// TIA Portal V18 export
// export: Created 2026-01-09T11:31:59.9051336Z, ExportSetting WithDefaults, DisplayName Totally Integrated Automation Portal, DisplayVersion V18 Update 5, DisplayName TIA Portal Openness, DisplayVersion V18 Update 5, DisplayName TIA Portal Teamcenter Gateway, DisplayVersion V18, DisplayName TIA Portal Version Control Interface, DisplayVersion V18, DisplayName SINAMICS Startdrive Advanced, DisplayVersion V18 SP2 Update 1, DisplayName SINAMICS Startdrive G110M, G120, G120C, G120D, G120P, G115D, DisplayVersion V18 SP2 Update 1, DisplayName SINAMICS Startdrive G130, G150, S120, S150, SINAMICS MV, S210, G220, S200, DisplayVersion V18 SP2 Update 1, DisplayName STEP 7 Professional, DisplayVersion V18 Update 5, DisplayName STEP 7 Safety, DisplayVersion V18, DisplayName WinCC Professional, DisplayVersion V18 Update 5
TagTable "1Command PLC To Mes_DB500"
  PLCtoMES_Load_Station1ChickInReq : Bool  (PLC tag PLCtoMES."PLC.Load_Station1ChickInReq", CPU S71500-2PN_TP700, 1 s)
  PLCtoMES_Load_Station2ChickInReq : Bool  (PLC tag PLCtoMES."PLC.Load_Station2ChickInReq", CPU S71500-2PN_TP700, 1 s)
  PLCtoMES_Load_Station3ChickInReq : Bool  (PLC tag PLCtoMES."PLC.Load_Station3ChickInReq", CPU S71500-2PN_TP700, 1 s)
  PLCtoMES_Load_Station4ChickInReq : Bool  (PLC tag PLCtoMES."PLC.Load_Station4ChickInReq", CPU S71500-2PN_TP700, 1 s)
  PLCtoMES_Load_Station5ChickInReq : Bool  (PLC tag PLCtoMES."PLC.Load_Station5ChickInReq", CPU S71500-2PN_TP700, 1 s)
  PLCtoMES_Load_Station6ChickInReq : Bool  (PLC tag PLCtoMES."PLC.Load_Station6ChickInReq", CPU S71500-2PN_TP700, 1 s)
  PLCtoMES_Load_Station7ChickInReq : Bool  (PLC tag PLCtoMES."PLC.Load_Station7ChickInReq", CPU S71500-2PN_TP700, 1 s)
  PLCtoMES_Load_Station8ChickInReq : Bool  (PLC tag PLCtoMES."PLC.Load_Station8ChickInReq", CPU S71500-2PN_TP700, 1 s)
  PLCtoMES_Load_SubPart1ChickInReq : Bool  (PLC tag PLCtoMES."PLC.Load_StoveCheckIn", CPU S71500-2PN_TP700, 1 s)
  PLCtoMES_Load_SubPart2ChickInReq : Bool  (PLC tag PLCtoMES.Spare_11, CPU S71500-2PN_TP700, 1 s)
  PLCtoMES_Load_SubPart3ChickInReq : Bool  (PLC tag PLCtoMES.Spare_12, CPU S71500-2PN_TP700, 1 s)
  PLCtoMES_Load_SubPart4ChickInReq : Bool  (PLC tag PLCtoMES.Spare_13, CPU S71500-2PN_TP700, 1 s)
  PLCtoMES_Load_SubPart5ChickInReq : Bool  (PLC tag PLCtoMES.Spare_14, CPU S71500-2PN_TP700, 1 s)
  PLCtoMES_Load_SubPart6ChickInReq : Bool  (PLC tag PLCtoMES.Spare_15, CPU S71500-2PN_TP700, 1 s)
  PLCtoMES_Load_SubPart7ChickInReq : Bool  (PLC tag PLCtoMES.Spare_16, CPU S71500-2PN_TP700, 1 s)
  PLCtoMES_Load_SubPart8ChickInReq : Bool  (PLC tag PLCtoMES.Spare_17, CPU S71500-2PN_TP700, 1 s)
  PLCtoMES_Load_Scanner1ChickInReq : Bool  (PLC tag PLCtoMES.Spare_18, CPU S71500-2PN_TP700, 1 s)
  PLCtoMES_Load_Scanner2ChickInReq : Bool  (PLC tag PLCtoMES.Spare_19, CPU S71500-2PN_TP700, 1 s)
  PLCtoMES_Load_Scanner3ChickInReq : Bool  (PLC tag PLCtoMES.Spare_20, CPU S71500-2PN_TP700, 1 s)
  PLCtoMES_Load_Scanner4ChickInReq : Bool  (PLC tag PLCtoMES.Spare_21, CPU S71500-2PN_TP700, 1 s)
  PLCtoMES_Load_Scanner5ChickInReq : Bool  (PLC tag PLCtoMES.Spare_22, CPU S71500-2PN_TP700, 1 s)
  PLCtoMES_Load_Scanner6ChickInReq : Bool  (PLC tag PLCtoMES.Spare_23, CPU S71500-2PN_TP700, 1 s)
  PLCtoMES_Load_Scanner7ChickInReq : Bool  (PLC tag PLCtoMES.Spare_24, CPU S71500-2PN_TP700, 1 s)
  PLCtoMES_Load_Scanner8ChickInReq : Bool  (PLC tag PLCtoMES.Spare_25, CPU S71500-2PN_TP700, 1 s)
  PLCtoMES_SpareByte : Byte  (PLC tag PLCtoMES.Spare_1, CPU S71500-2PN_TP700, 1 s)
  PLCtoMES_Load_PrintReq : Bool  (PLC tag PLCtoMES.Spare_2, CPU S71500-2PN_TP700, 1 s)
  PLCtoMES_Load_DataMatrixCheckReq : Bool  (PLC tag PLCtoMES.Spare_3, CPU S71500-2PN_TP700, 1 s)
  PLCtoMES_Load_Spare : Bool  (PLC tag PLCtoMES.Spare_4, CPU S71500-2PN_TP700, 1 s)
  PLCtoMES_Load_Spare_1 : Bool  (PLC tag PLCtoMES.Spare_5, CPU S71500-2PN_TP700, 1 s)
  PLCtoMES_Load_Spare_2 : Bool  (PLC tag PLCtoMES.Spare_6, CPU S71500-2PN_TP700, 1 s)
  PLCtoMES_Load_Spare_3 : Bool  (PLC tag PLCtoMES.Spare_7, CPU S71500-2PN_TP700, 1 s)
  PLCtoMES_Load_Spare_4 : Bool  (PLC tag PLCtoMES.Spare_8, CPU S71500-2PN_TP700, 1 s)
  PLCtoMES_Load_Spare_5 : Bool  (PLC tag PLCtoMES.Spare_9, CPU S71500-2PN_TP700, 1 s)
  PLCtoMES_Unload_Station1DataSaveReq : Bool  (PLC tag PLCtoMES.Static_2, CPU S71500-2PN_TP700, 1 s)
  PLCtoMES_Unload_Station2DataSaveReq : Bool  (PLC tag PLCtoMES."PLC.Unload_Station1DataSaveReq", CPU S71500-2PN_TP700, 1 s)
  PLCtoMES_Unload_Station3DataSaveReq : Bool  (PLC tag PLCtoMES."PLC.Unload_Station2DataSaveReq", CPU S71500-2PN_TP700, 1 s)
  PLCtoMES_Unload_Station4DataSaveReq : Bool  (PLC tag PLCtoMES."PLC.Unload_Station3DataSaveReq", CPU S71500-2PN_TP700, 1 s)
  PLCtoMES_Unload_Station5DataSaveReq : Bool  (PLC tag PLCtoMES."PLC.Unload_Station4DataSaveReq", CPU S71500-2PN_TP700, 1 s)
  PLCtoMES_Unload_Station6DataSaveReq : Bool  (PLC tag PLCtoMES."PLC.Unload_Station5DataSaveReq", CPU S71500-2PN_TP700, 1 s)
  PLCtoMES_Unload_Station7DataSaveReq : Bool  (PLC tag PLCtoMES."PLC.Unload_Station6DataSaveReq", CPU S71500-2PN_TP700, 1 s)
  PLCtoMES_Unload_Station8DataSaveReq : Bool  (PLC tag PLCtoMES."PLC.Unload_Station7DataSaveReq", CPU S71500-2PN_TP700, 1 s)
  PLCtoMES_P-HeartBeat : Bool  (PLC tag PLCtoMES."PLC.Unload_Station8DataSaveReq", CPU S71500-2PN_TP700, 1 s)
